Fanuc KAREL source: kt00911.KL

PROGRAM KT00911
%STACKSIZE=65535
%PRIORITY=65535
%NOLOCKGROUP
VAR
P1 : JOINTPOS9
P2 : JOINTPOS9
-- UNRESOLVED DECLARATIONS (source type spelling not recovered)
-- OUT : TYPE_0x0013 (type_u16=0x0013)
BEGIN
-- UNSAFE_SOURCE_IR line 9: OUT = ORIENT(convert_jointpos9_to_position(P1))
END KT00911
